Omron Sysmac Studio project 2.0_integration_1 (Sysmac Studio 1.54.0.64019, StandardProject)

# Controller new_Controller_0: NJ301-1100 version 1.14
Units and slaves: Node1 : NX-ECC201 (E001); Unit 1 : NX-PC0020 (N1); Unit 2 : NX-ID5442 (N2); Unit 3 : NX-PC0010 (N3); Unit 4 : NX-PC0020 (N4); Unit 5 : NX-OD5121 (N5); Unit 6 : NX-PC0010 (N6); Power Supply : NJ-Px3001; CPU : NJ301-1100; 0 [Unit 0] : CJ1W-AD041-V1 (J01); 1 [Unit 1] : CJ1W-DA041 (J02); 2 : CJ1W-ID211 (J03); 3 : CJ1W-OC211 (J04)
Task PrimaryTask (priority 4, period or condition 1000): Program0

VAR_GLOBAL
    Station_1B2 : BOOL;  (* Lifting Cylinder Down; at IOBus://rack#0/slot#2/Ch1_In/Ch1_In05; published *)
    Station_1B1 : BOOL;  (* Lifting Cylinder Up; at IOBus://rack#0/slot#2/Ch1_In/Ch1_In04; published *)
    Station_B5 : BOOL;  (* Workpiece Height Correct; at IOBus://rack#0/slot#2/Ch1_In/Ch1_In03; published *)
    Station_3S1 : BOOL;  (* arm_in_magazine; published *)
    Station_3S2 : BOOL;  (* arm_in_downstream; published *)
    Station_2B1 : BOOL;  (* Ejecting Cylinder Retracted; at IOBus://rack#0/slot#2/Ch1_In/Ch1_In06; published *)
    Panel_S1 : BOOL;  (* start_button; at IOBus://rack#0/slot#2/Ch1_In/Ch1_In08; published *)
    Panel_S2 : BOOL;  (* stop_button; at IOBus://rack#0/slot#2/Ch1_In/Ch1_In09; published *)
    Panel_S4 : BOOL;  (* reset_button; at IOBus://rack#0/slot#2/Ch1_In/Ch1_In11; published *)
    Station_1Y1 : BOOL;  (* Lift Down; at IOBus://rack#0/slot#3/Ch1_Out/Ch1_Out00; published *)
    Station_1Y2 : BOOL;  (* Lift Up; at IOBus://rack#0/slot#3/Ch1_Out/Ch1_Out01; published *)
    Station_2Y1 : BOOL;  (* Advance Ejecting Cylinder; at IOBus://rack#0/slot#3/Ch1_Out/Ch1_Out02; published *)
    Station_3Y1 : BOOL;  (* Air Cushion On; at IOBus://rack#0/slot#3/Ch1_Out/Ch1_Out03; published *)
    Station_3Y2 : BOOL;  (* arm_2_downstream; published *)
    Station_H1 : BOOL;  (* start light; at IOBus://rack#0/slot#3/Ch1_Out/Ch1_Out08; published *)
    Station_H2 : BOOL;  (* reset light; at IOBus://rack#0/slot#3/Ch1_Out/Ch1_Out09; published *)
    Panel_H3 : BOOL;  (* Q1 light; at IOBus://rack#0/slot#3/Ch1_Out/Ch1_Out10; published *)
    Panel_H4 : BOOL;  (* Q2 light; at IOBus://rack#0/slot#3/Ch1_Out/Ch1_Out11; published *)
    Station_1B1_in : BOOL;
    IP_FI : BOOL;  (* Succeeding Station Free; at IOBus://rack#0/slot#2/Ch1_In/Ch1_In07 *)
    Part_AV : BOOL;  (* Workpiece Available; at IOBus://rack#0/slot#2/Ch1_In/Ch1_In00 *)
    Station_B2 : BOOL;  (* Workpiece not black; at IOBus://rack#0/slot#2/Ch1_In/Ch1_In01 *)
    Station_B4 : BOOL;  (* Safety Through Beam; at IOBus://rack#0/slot#2/Ch1_In/Ch1_In02 *)
    IP_N_FO : BOOL;  (* Station Occupied; at IOBus://rack#0/slot#3/Ch1_Out/Ch1_Out07 *)
END_VAR

PROGRAM Program0
VAR
    FB_Panel_1 : FB_Panel;
    run_mode : BOOL;
    stop_mode : BOOL;
    reset_mode : BOOL;
    FB_Actuator_T1_1 : FB_Actuator_T1;
    timer_t1 : TON;
    error_mode : BOOL;
    FB_Actuator_T2_1 : FB_Actuator_T2;
    Piston : RS;
    error_ejec : BOOL;
    extend_piston : BOOL;
    workpiece_ready_set : BOOL;
    flip_flop_1 : RS;
    workpiece_ready : BOOL;
    workpiece_picked_up : BOOL;
    wait_for_piston : TON;
    Workpiece_Checker_1 : Workpiece_Checker;
    error_state : BOOL;
    error_suction : BOOL;
    error_t1 : BOOL;
    error_t2 : BOOL;
    rs1 : RS;
    rs2 : RS;
    rs3 : RS;
    e1 : BOOL;
    e2 : BOOL;
    e3 : BOOL;
    error_lift : BOOL;
    Control_T1_1 : Control_T1;
    error_q2_out : BOOL;
    Station_h3 : BOOL;
    Station_h4 : BOOL;
    FB_Receiver_1 : FB_Receiver;
    start_reciever : BOOL;
    stop_reciever : BOOL;
    reset_reciever : BOOL;
    next_ready : BOOL;
    start_button : BOOL;
    stop_button : BOOL;
    reset_button : BOOL;
    FB_Sender_1 : FB_Sender;
    need_piece : BOOL;
END_VAR
VAR_EXTERNAL
    Station_3S1 : BOOL;
    Panel_S2 : BOOL;
    Station_3Y2 : BOOL;
    Station_3S2 : BOOL;
    Panel_S1 : BOOL;
    Station_3Y1 : BOOL;
    Panel_S4 : BOOL;
    Station_H1 : BOOL;
    Station_H2 : BOOL;
    Panel_H4 : BOOL;
    Panel_H3 : BOOL;
    Station_1B2 : BOOL;
    Station_1B1 : BOOL;
    Station_1Y1 : BOOL;
    Station_2Y1 : BOOL;
    Station_2B1 : BOOL;
    Station_B4 : BOOL;
    Station_1Y2 : BOOL;
    Station_B2 : BOOL;
    Part_AV : BOOL;
    Station_B5 : BOOL;
    IP_FI : BOOL;
    IP_N_FO : BOOL;
END_VAR

(* Section Section0: ladder, written here as Structured Text *)

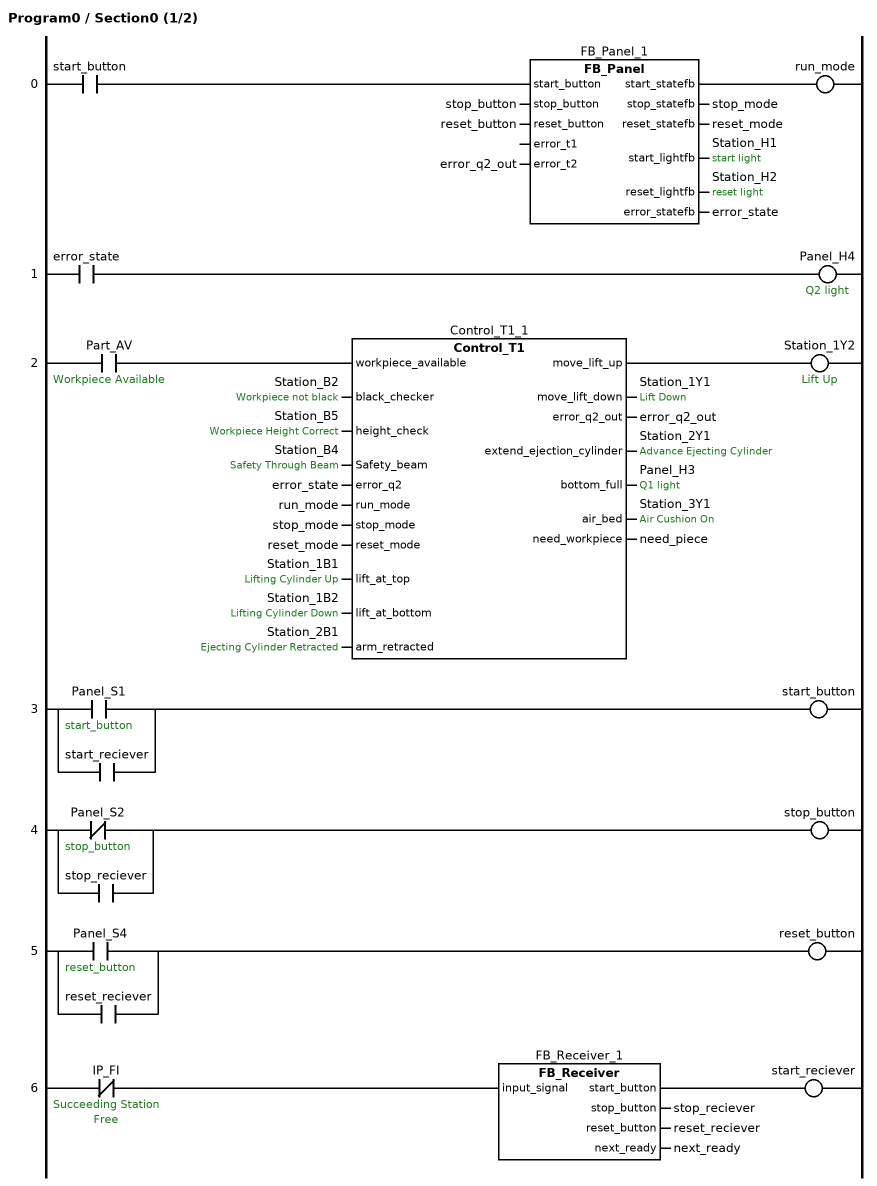
(* Rung 0 *)
FB_Panel_1(start_button := start_button, stop_button := stop_button, reset_button := reset_button, error_t2 := error_q2_out, stop_statefb => stop_mode, reset_statefb => reset_mode, start_lightfb => Station_H1, reset_lightfb => Station_H2, error_statefb => error_state);
run_mode := FB_Panel_1.start_statefb;
(* Rung 1 *)
Panel_H4 := error_state;
(* Rung 2 *)
Control_T1_1(workpiece_available := Part_AV, black_checker := Station_B2, height_check := Station_B5, Safety_beam := Station_B4, error_q2 := error_state, run_mode := run_mode, stop_mode := stop_mode, reset_mode := reset_mode, lift_at_top := Station_1B1, lift_at_bottom := Station_1B2, arm_retracted := Station_2B1, move_lift_down => Station_1Y1, error_q2_out => error_q2_out, extend_ejection_cylinder => Station_2Y1, bottom_full => Panel_H3, air_bed => Station_3Y1, need_workpiece => need_piece);
Station_1Y2 := Control_T1_1.move_lift_up;
(* Rung 3 *)
start_button := Panel_S1 OR start_reciever;
(* Rung 4 *)
stop_button := NOT Panel_S2 OR stop_reciever;
(* Rung 5 *)
reset_button := Panel_S4 OR reset_reciever;
(* Rung 6 *)
FB_Receiver_1(input_signal := NOT IP_FI, stop_button => stop_reciever, reset_button => reset_reciever, next_ready => next_ready);
start_reciever := FB_Receiver_1.start_button;

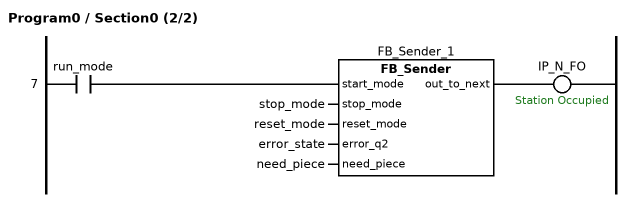
(* Rung 7 *)
FB_Sender_1(start_mode := run_mode, stop_mode := stop_mode, reset_mode := reset_mode, error_q2 := error_state, need_piece := need_piece);
IP_N_FO := FB_Sender_1.out_to_next;
END_PROGRAM

FUNCTION_BLOCK FB_Panel
VAR
    flip_flop : RS;
    flip_flop2 : RS;
    flip_flop_3 : RS;
    flip_flop3 : RS;
    stop_or_error : BOOL;
    error_q2 : BOOL;
    flip_flop4 : RS;
END_VAR
VAR_OUTPUT
    start_statefb : BOOL;
    stop_statefb : BOOL;
    reset_statefb : BOOL;
END_VAR
VAR_INPUT
    start_button : BOOL := False;
    stop_button : BOOL := False;
    reset_button : BOOL := False;
END_VAR
VAR_OUTPUT
    start_lightfb : BOOL;
    reset_lightfb : BOOL;
    error_statefb : BOOL;
END_VAR
VAR_INPUT
    error_t1 : BOOL;
    error_t2 : BOOL;
END_VAR
VAR_EXTERNAL
    Panel_H4 : BOOL;
END_VAR
(* ladder, written here as Structured Text *)

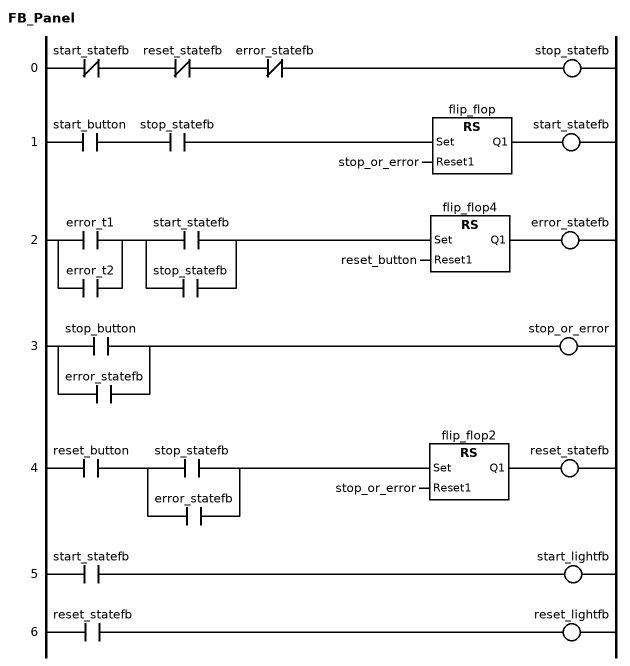
(* Rung 0 *)
stop_statefb := NOT start_statefb AND NOT reset_statefb AND NOT error_statefb;
(* Rung 1 *)
flip_flop(Set := start_button AND stop_statefb, Reset1 := stop_or_error);
start_statefb := flip_flop.Q1;
(* Rung 2 *)
flip_flop4(Set := (error_t1 OR error_t2) AND (start_statefb OR stop_statefb), Reset1 := reset_button);
error_statefb := flip_flop4.Q1;
(* Rung 3 *)
stop_or_error := stop_button OR error_statefb;
(* Rung 4 *)
flip_flop2(Set := reset_button AND (stop_statefb OR error_statefb), Reset1 := stop_or_error);
reset_statefb := flip_flop2.Q1;
(* Rung 5 *)
start_lightfb := start_statefb;
(* Rung 6 *)
reset_lightfb := reset_statefb;
END_FUNCTION_BLOCK

FUNCTION_BLOCK FB_Actuator_T2
VAR
    reset_to_home : BOOL;
    retract_ff : RS;
    extend_ff : RS;
    extend_t : TON;
    retract_t : TON;
    retract_err : BOOL;
    extend_err : BOOL;
    workpiece_lifted : BOOL;
    Workpiece_ejection : RS;
END_VAR
VAR_INPUT
    run_mode : BOOL;
    reset_mode : BOOL;
    stop_mode : BOOL;
    error_mode : BOOL;
END_VAR
VAR_OUTPUT
    retract_piston : BOOL;
    extend_piston : BOOL;
END_VAR
VAR_INPUT
    piston_retracted : BOOL;
    piston_extended : BOOL;
END_VAR
VAR_OUTPUT
    error_eject : BOOL;
END_VAR
VAR_INPUT
    Workpiece_ready : BOOL;
END_VAR
VAR_OUTPUT
    Mag_Empty_out : BOOL;
END_VAR
VAR_INPUT
    Mag_state : BOOL;
END_VAR
VAR_EXTERNAL
    Station_B4 : BOOL;
    Station_1B1 : BOOL;
    Station_1B2 : BOOL;
    Station_2Y1 : BOOL;
END_VAR
(* ladder, written here as Structured Text *)

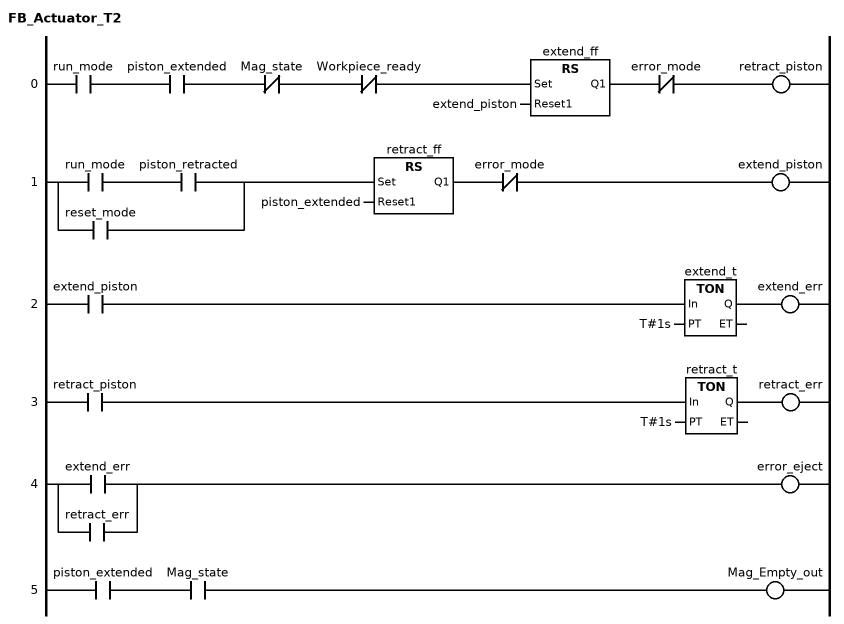
(* Rung 0 *)
extend_ff(Set := run_mode AND piston_extended AND NOT Mag_state AND NOT Workpiece_ready, Reset1 := extend_piston);
retract_piston := extend_ff.Q1 AND NOT error_mode;
(* Rung 1 *)
retract_ff(Set := (run_mode AND piston_retracted) OR reset_mode, Reset1 := piston_extended);
extend_piston := retract_ff.Q1 AND NOT error_mode;
(* Rung 2 *)
extend_t(In := extend_piston, PT := T#1s);
extend_err := extend_t.Q;
(* Rung 3 *)
retract_t(In := retract_piston, PT := T#1s);
retract_err := retract_t.Q;
(* Rung 4 *)
error_eject := extend_err OR retract_err;
(* Rung 5 *)
Mag_Empty_out := piston_extended AND Mag_state;
END_FUNCTION_BLOCK

FUNCTION_BLOCK Workpiece_Checker
VAR
    wait_for_piston : TON;
    flip_flop_1 : RS;
    workpiece_not_ready : BOOL;
END_VAR
VAR_INPUT
    reset_state : BOOL;
    workpiece_ready_set : BOOL;
    workpiece_picked_up : BOOL (* edge DownDirection *);
END_VAR
VAR_OUTPUT
    workpiece_ready : BOOL;
END_VAR
(* ladder, written here as Structured Text *)

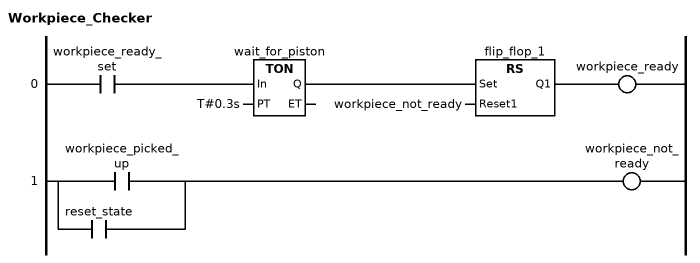
(* Rung 0 *)
wait_for_piston(In := workpiece_ready_set, PT := T#0.3s);
flip_flop_1(Set := wait_for_piston.Q, Reset1 := workpiece_not_ready);
workpiece_ready := flip_flop_1.Q1;
(* Rung 1 *)
workpiece_not_ready := workpiece_picked_up OR reset_state;
END_FUNCTION_BLOCK

FUNCTION_BLOCK FB_Actuator_T1
VAR
    flip_flop_1 : RS;
    flip_flop_2 : RS;
    reset_to_home : BOOL;
    timer_t1 : TON;
    flip_flop_3 : RS;
    timer_t2 : TON;
    flip_flop_4 : RS;
    error_toSub : BOOL;
    error_toHome : BOOL;
    middle_timer : AccumulationTimer;
    flip_flop_5 : RS;
    reset_middle : BOOL;
    flip_flop6 : RS;
    move_to_middle_from_home : BOOL;
    move_to_home : BOOL;
    move_to_middle_from_sub : BOOL;
    unknown_pos : BOOL;
    reset_vac_arm_to_sub : BOOL;
    timer_t3 : TON;
    t : TIME;
    unknown_pos_timer : TON;
    TOF_1 : TOF;
    move_to_sub : BOOL;
END_VAR
VAR_INPUT
    Arm_In_Mag_Pos : BOOL;
    Arm_In_Sub_Pos : BOOL;
    stop_mode : BOOL;
END_VAR
VAR_OUTPUT
    error_arm : BOOL;
    arm_to_sub : BOOL;
    arm_to_home : BOOL;
END_VAR
VAR_INPUT
    error_q2 : BOOL;
    set_move_to_sub : BOOL;
    set_move_to_home : BOOL;
    set_move_to_middle_from_home : BOOL;
    set_move_to_middle_from_sub : BOOL;
END_VAR
VAR_OUTPUT
    middle_pos : BOOL;
END_VAR
VAR_INPUT
    reset_mode : BOOL;
END_VAR
VAR_EXTERNAL
    Station_1B1 : BOOL;
END_VAR
(* ladder, written here as Structured Text *)

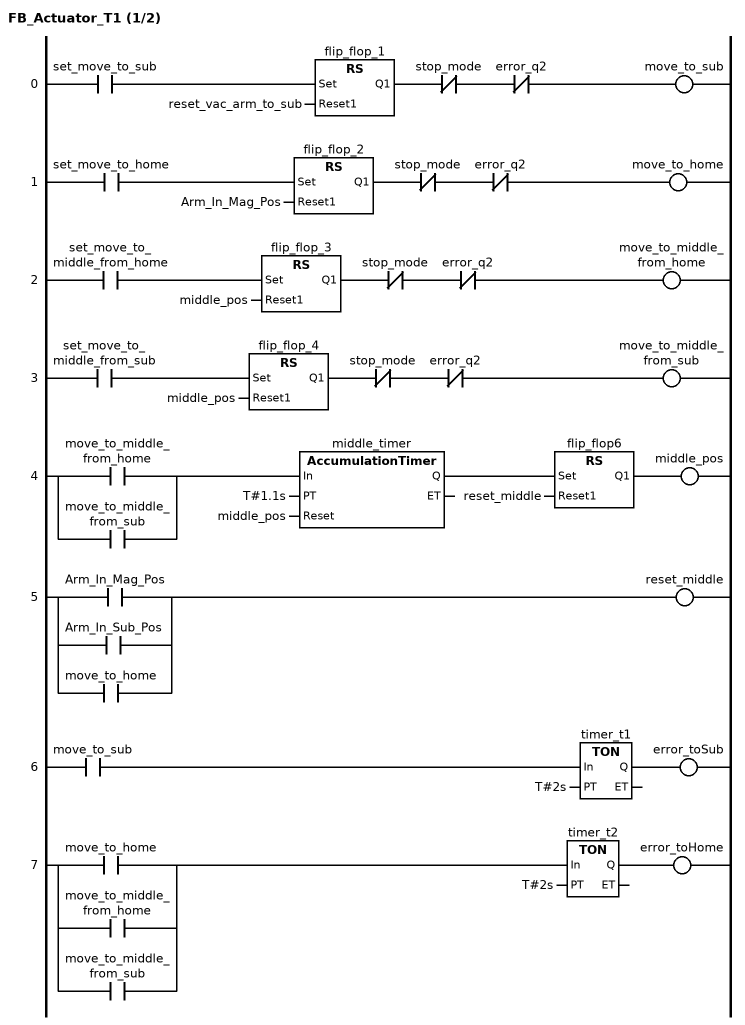
(* Rung 0 *)
flip_flop_1(Set := set_move_to_sub, Reset1 := reset_vac_arm_to_sub);
move_to_sub := flip_flop_1.Q1 AND NOT stop_mode AND NOT error_q2;
(* Rung 1 *)
flip_flop_2(Set := set_move_to_home, Reset1 := Arm_In_Mag_Pos);
move_to_home := flip_flop_2.Q1 AND NOT stop_mode AND NOT error_q2;
(* Rung 2 *)
flip_flop_3(Set := set_move_to_middle_from_home, Reset1 := middle_pos);
move_to_middle_from_home := flip_flop_3.Q1 AND NOT stop_mode AND NOT error_q2;
(* Rung 3 *)
flip_flop_4(Set := set_move_to_middle_from_sub, Reset1 := middle_pos);
move_to_middle_from_sub := flip_flop_4.Q1 AND NOT stop_mode AND NOT error_q2;
(* Rung 4 *)
middle_timer(In := move_to_middle_from_home OR move_to_middle_from_sub, PT := T#1.1s, Reset := middle_pos);
flip_flop6(Set := middle_timer.Q, Reset1 := reset_middle);
middle_pos := flip_flop6.Q1;
(* Rung 5 *)
reset_middle := Arm_In_Mag_Pos OR Arm_In_Sub_Pos OR move_to_home;
(* Rung 6 *)
timer_t1(In := move_to_sub, PT := T#2s);
error_toSub := timer_t1.Q;
(* Rung 7 *)
timer_t2(In := move_to_home OR move_to_middle_from_home OR move_to_middle_from_sub, PT := T#2s);
error_toHome := timer_t2.Q;

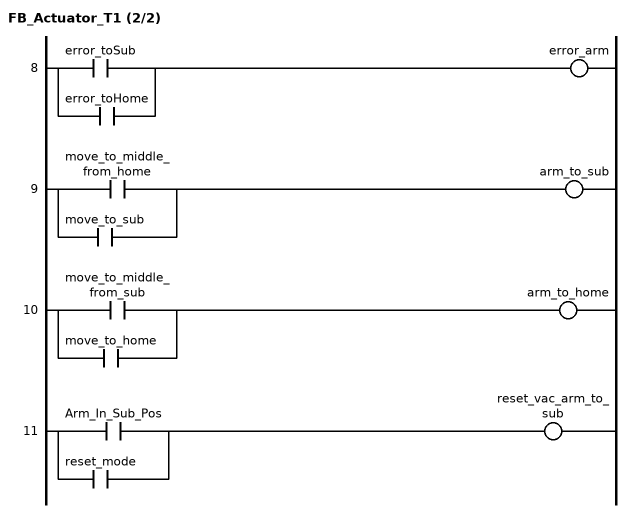
(* Rung 8 *)
error_arm := error_toSub OR error_toHome;
(* Rung 9 *)
arm_to_sub := move_to_middle_from_home OR move_to_sub;
(* Rung 10 *)
arm_to_home := move_to_middle_from_sub OR move_to_home;
(* Rung 11 *)
reset_vac_arm_to_sub := Arm_In_Sub_Pos OR reset_mode;
END_FUNCTION_BLOCK

FUNCTION_BLOCK Control_T1
VAR
    FB_Actuator_T1_1 : FB_Actuator_T1;
    set_move_lift_down : BOOL;
    set_move_lift_up : BOOL;
    lift_moved : BOOL;
    lift_move_rs : RS;
    wait_lift : BOOL;
    wait_t3_up : TON;
    wait_t3_down : TON;
    error_t3 : BOOL;
    error_lift : BOOL;
    reset_safety_beam : BOOL;
    Safety_beam_error_1 : BOOL;
    safety_timer : TON;
    Safety_beam_error_2 : BOOL;
    safet_beam_counter : CTU;
    safety_beam_error : BOOL;
    cnt : INT;
    TOF_safety_beam : TOF;
    safetybeam_TON : TON;
    t3_finished : BOOL;
    rs_output_top : RS;
    rs_output_bottom : RS;
    bottom_eject_counter : CTU;
    eject_top : BOOL;
    eject_bot : BOOL;
    reset_t3_ejector : BOOL;
    eject_bot_timer : TON;
    cnt2 : INT;
    actuator_T3 : BOOL;
    workpiece_carried_rs : RS;
    workpiece_carried : BOOL;
    cycle_complete : BOOL;
    reset_workpiece_carried : BOOL;
    r_trig_t3_cycle : R_TRIG;
    wait_lift_down : TON;
    eject_top_timer : TON;
    error_no_room_bottom : BOOL;
    rs_white_piece : RS;
    white_eject_bottom : BOOL;
    wait_lift_up : TON;
    rs_test_whiteandfull : RS;
    q2_full_bottom : BOOL;
    pulse_time_air_bed : TP;
    Control_T3_1 : control_T3;
    rs_error_t3 : RS;
    rs_error_safety_beam : RS;
    rs_error_lift : RS;
    test_error_t3 : BOOL;
    test_error_beam : BOOL;
    test_error_lift : BOOL;
    rs_bottom_full_error : RS;
    test_error_bottom : BOOL;
    TON_error_no_room_bottom : TON;
    delay_white_top : TON;
    reset_workpiece_carried_TP : TP;
    wait_T3 : CTU;
    cnt_actuator : INT;
    wait_workpiece_carried_TON : TON;
    request_workpiece_TON : TON;
END_VAR
VAR_INPUT
    workpiece_available : BOOL;
    black_checker : BOOL;
    height_check : BOOL;
    Safety_beam : BOOL;
    error_q2 : BOOL;
    run_mode : BOOL;
    stop_mode : BOOL;
    reset_mode : BOOL;
    lift_at_top : BOOL;
    lift_at_bottom : BOOL;
END_VAR
VAR_OUTPUT
    move_lift_up : BOOL;
    move_lift_down : BOOL;
    error_q2_out : BOOL;
    extend_ejection_cylinder : BOOL;
END_VAR
VAR_INPUT
    arm_retracted : BOOL;
END_VAR
VAR_OUTPUT
    bottom_full : BOOL;
    air_bed : BOOL;
    need_workpiece : BOOL;
END_VAR
VAR_EXTERNAL
    Station_1B1 : BOOL;
    Station_1B1_in : BOOL;
    Station_1B2 : BOOL;
    Station_B2 : BOOL;
END_VAR
VAR
    _e1 : R_TRIG;
    _e2 : R_TRIG;
END_VAR
(* ladder, written here as Structured Text *)

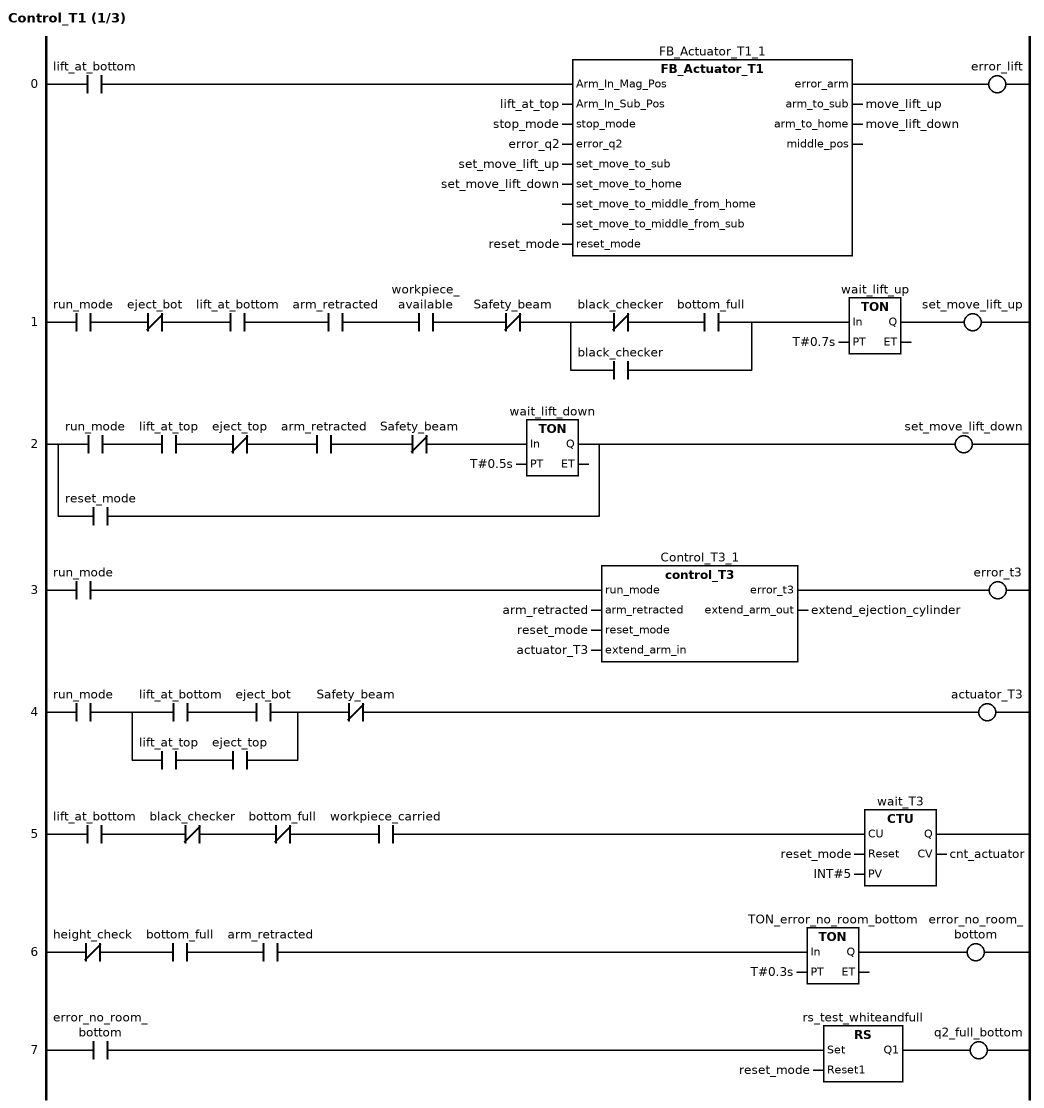
(* Rung 0 *)
FB_Actuator_T1_1(Arm_In_Mag_Pos := lift_at_bottom, Arm_In_Sub_Pos := lift_at_top, stop_mode := stop_mode, error_q2 := error_q2, set_move_to_sub := set_move_lift_up, set_move_to_home := set_move_lift_down, reset_mode := reset_mode, arm_to_sub => move_lift_up, arm_to_home => move_lift_down);
error_lift := FB_Actuator_T1_1.error_arm;
(* Rung 1 *)
wait_lift_up(In := run_mode AND NOT eject_bot AND lift_at_bottom AND arm_retracted AND workpiece_available AND NOT Safety_beam AND ((NOT black_checker AND bottom_full) OR black_checker), PT := T#0.7s);
set_move_lift_up := wait_lift_up.Q;
(* Rung 2 *)
wait_lift_down(In := run_mode AND lift_at_top AND NOT eject_top AND arm_retracted AND NOT Safety_beam, PT := T#0.5s);
set_move_lift_down := wait_lift_down.Q OR reset_mode;
(* Rung 3 *)
Control_T3_1(run_mode := run_mode, arm_retracted := arm_retracted, reset_mode := reset_mode, extend_arm_in := actuator_T3, extend_arm_out => extend_ejection_cylinder);
error_t3 := Control_T3_1.error_t3;
(* Rung 4 *)
actuator_T3 := run_mode AND ((lift_at_bottom AND eject_bot) OR (lift_at_top AND eject_top)) AND NOT Safety_beam;
(* Rung 5 *)
_e1(CLK := lift_at_bottom AND NOT black_checker AND NOT bottom_full AND workpiece_carried);
wait_T3(CU := _e1.Q, Reset := reset_mode, PV := INT#5, CV => cnt_actuator);
(* Rung 6 *)
TON_error_no_room_bottom(In := NOT height_check AND bottom_full AND arm_retracted, PT := T#0.3s);
error_no_room_bottom := TON_error_no_room_bottom.Q;
(* Rung 7 *)
rs_test_whiteandfull(Set := error_no_room_bottom, Reset1 := reset_mode);
q2_full_bottom := rs_test_whiteandfull.Q1;

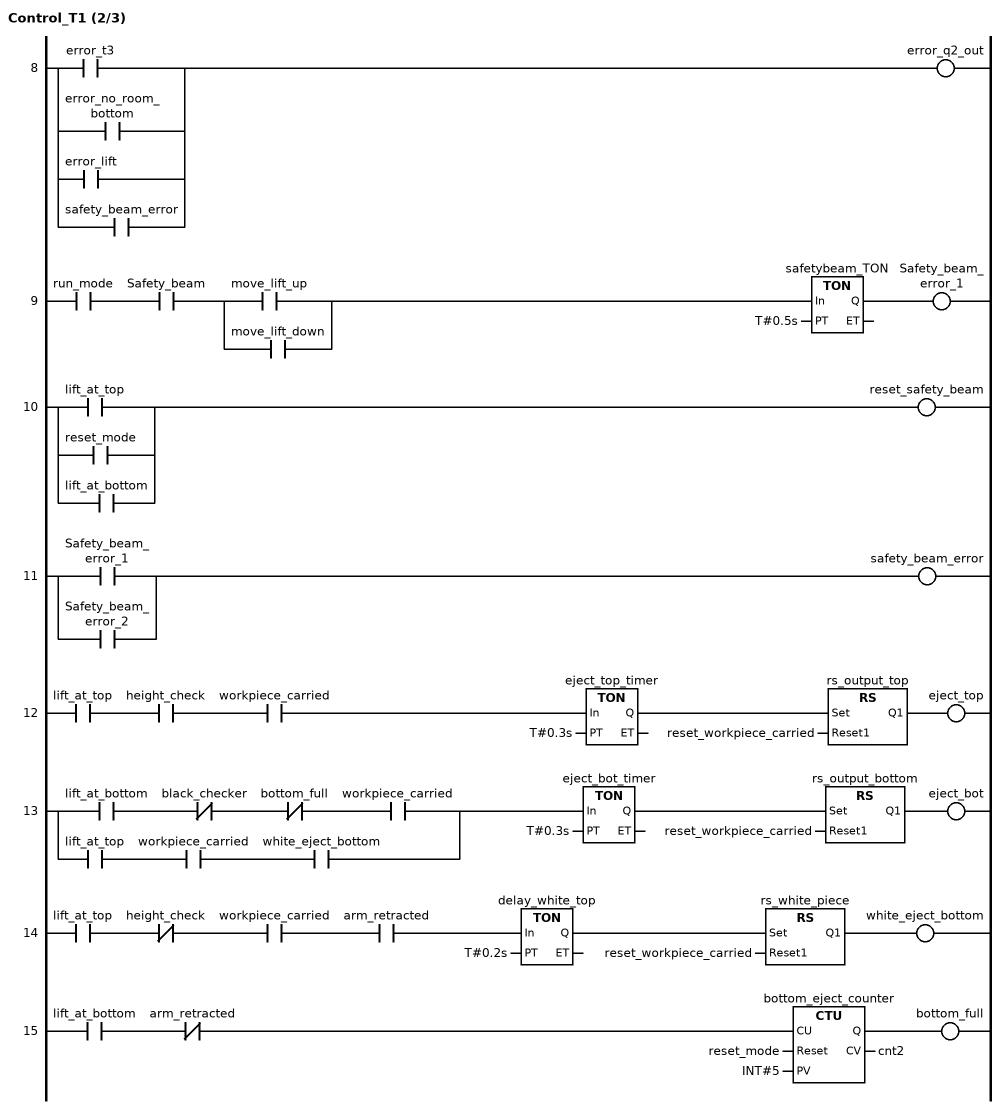
(* Rung 8 *)
error_q2_out := error_t3 OR error_no_room_bottom OR error_lift OR safety_beam_error;
(* Rung 9 *)
safetybeam_TON(In := run_mode AND Safety_beam AND (move_lift_up OR move_lift_down), PT := T#0.5s);
Safety_beam_error_1 := safetybeam_TON.Q;
(* Rung 10 *)
reset_safety_beam := lift_at_top OR reset_mode OR lift_at_bottom;
(* Rung 11 *)
safety_beam_error := Safety_beam_error_1 OR Safety_beam_error_2;
(* Rung 12 *)
eject_top_timer(In := lift_at_top AND height_check AND workpiece_carried, PT := T#0.3s);
rs_output_top(Set := eject_top_timer.Q, Reset1 := reset_workpiece_carried);
eject_top := rs_output_top.Q1;
(* Rung 13 *)
eject_bot_timer(In := (lift_at_bottom AND NOT black_checker AND NOT bottom_full AND workpiece_carried) OR (lift_at_top AND workpiece_carried AND white_eject_bottom), PT := T#0.3s);
rs_output_bottom(Set := eject_bot_timer.Q, Reset1 := reset_workpiece_carried);
eject_bot := rs_output_bottom.Q1;
(* Rung 14 *)
delay_white_top(In := lift_at_top AND NOT height_check AND workpiece_carried AND arm_retracted, PT := T#0.2s);
rs_white_piece(Set := delay_white_top.Q, Reset1 := reset_workpiece_carried);
white_eject_bottom := rs_white_piece.Q1;
(* Rung 15 *)
_e2(CLK := lift_at_bottom AND NOT arm_retracted);
bottom_eject_counter(CU := _e2.Q, Reset := reset_mode, PV := INT#5, CV => cnt2);
bottom_full := bottom_eject_counter.Q;

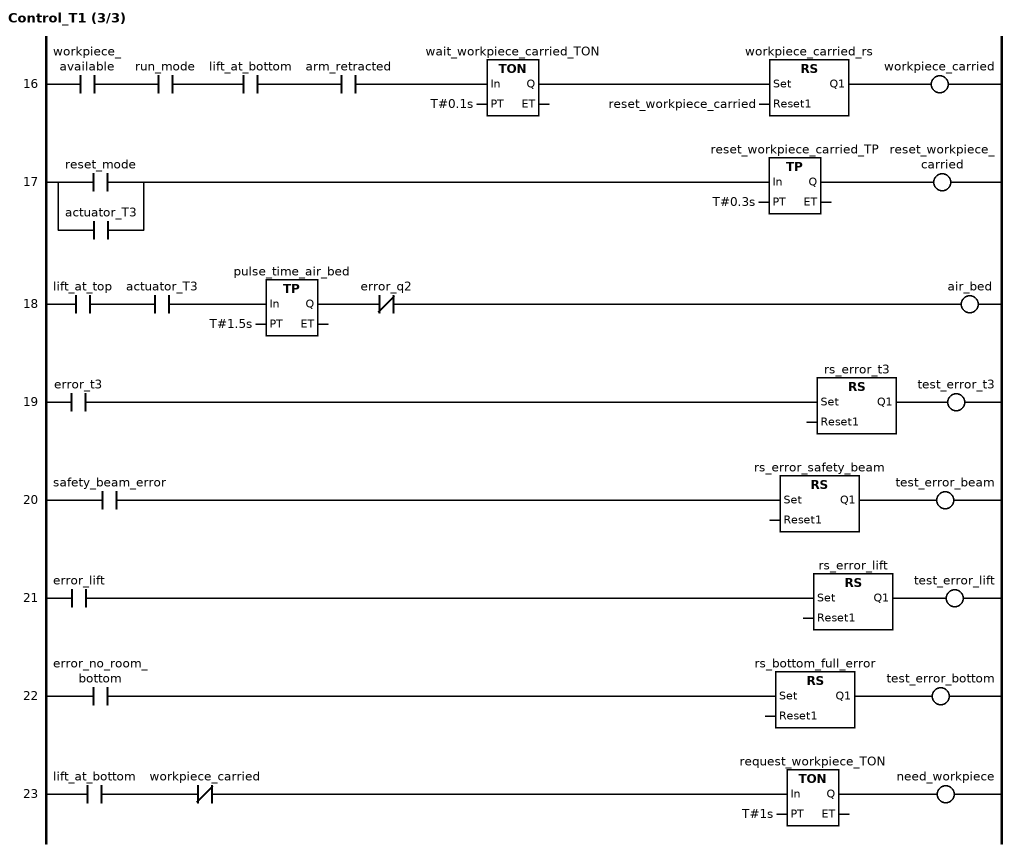
(* Rung 16 *)
wait_workpiece_carried_TON(In := workpiece_available AND run_mode AND lift_at_bottom AND arm_retracted, PT := T#0.1s);
workpiece_carried_rs(Set := wait_workpiece_carried_TON.Q, Reset1 := reset_workpiece_carried);
workpiece_carried := workpiece_carried_rs.Q1;
(* Rung 17 *)
reset_workpiece_carried_TP(In := reset_mode OR actuator_T3, PT := T#0.3s);
reset_workpiece_carried := reset_workpiece_carried_TP.Q;
(* Rung 18 *)
pulse_time_air_bed(In := lift_at_top AND actuator_T3, PT := T#1.5s);
air_bed := pulse_time_air_bed.Q AND NOT error_q2;
(* Rung 19 *)
rs_error_t3(Set := error_t3);
test_error_t3 := rs_error_t3.Q1;
(* Rung 20 *)
rs_error_safety_beam(Set := safety_beam_error);
test_error_beam := rs_error_safety_beam.Q1;
(* Rung 21 *)
rs_error_lift(Set := error_lift);
test_error_lift := rs_error_lift.Q1;
(* Rung 22 *)
rs_bottom_full_error(Set := error_no_room_bottom);
test_error_bottom := rs_bottom_full_error.Q1;
(* Rung 23 *)
request_workpiece_TON(In := lift_at_bottom AND NOT workpiece_carried, PT := T#1s);
need_workpiece := request_workpiece_TON.Q;
END_FUNCTION_BLOCK

FUNCTION_BLOCK FB_Actuator_T3
VAR
    TOF_1 : TOF;
    extend_arm_error_rs : RS;
    extend_arm_error_TON : TON;
    retract_arm : BOOL;
    Error_held_timer : AccumulationTimer;
    arm_extended_out : BOOL;
    reset_timer : BOOL;
    arm_out_timer : TON;
    arm_out_rs : RS;
    arm_extended_rs : RS;
    cycle_check_rs : RS;
    error_t3_1 : BOOL;
END_VAR
VAR_INPUT
    extend_arm_in : BOOL;
END_VAR
VAR_OUTPUT
    extend_arm_out : BOOL;
END_VAR
VAR_INPUT
    run_mode : BOOL;
    arm_retracted : BOOL;
END_VAR
VAR_OUTPUT
    error_t3 : BOOL;
END_VAR
VAR_INPUT
    reset_mode : BOOL;
    retract_arm_command : BOOL;
END_VAR
VAR_OUTPUT
    arm_extended : BOOL;
END_VAR
(* ladder, written here as Structured Text *)

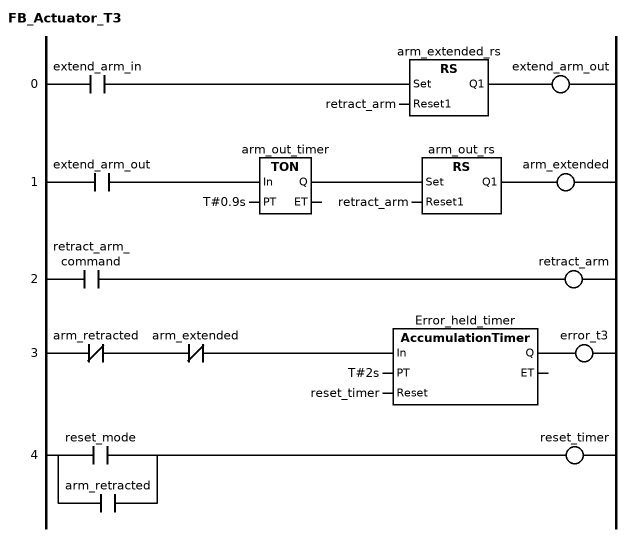
(* Rung 0 *)
arm_extended_rs(Set := extend_arm_in, Reset1 := retract_arm);
extend_arm_out := arm_extended_rs.Q1;
(* Rung 1 *)
arm_out_timer(In := extend_arm_out, PT := T#0.9s);
arm_out_rs(Set := arm_out_timer.Q, Reset1 := retract_arm);
arm_extended := arm_out_rs.Q1;
(* Rung 2 *)
retract_arm := retract_arm_command;
(* Rung 3 *)
Error_held_timer(In := NOT arm_retracted AND NOT arm_extended, PT := T#2s, Reset := reset_timer);
error_t3 := Error_held_timer.Q;
(* Rung 4 *)
reset_timer := reset_mode OR arm_retracted;
END_FUNCTION_BLOCK

FUNCTION_BLOCK control_T3
VAR
    FB_Actuator_T3_2 : FB_Actuator_T3;
    retract_arm : BOOL;
    arm_extended : BOOL;
    extend_arm_command : BOOL;
END_VAR
VAR_INPUT
    run_mode : BOOL;
    arm_retracted : BOOL;
    reset_mode : BOOL;
END_VAR
VAR_OUTPUT
    error_t3 : BOOL;
    extend_arm_out : BOOL;
END_VAR
VAR_INPUT
    extend_arm_in : BOOL;
END_VAR
(* ladder, written here as Structured Text *)

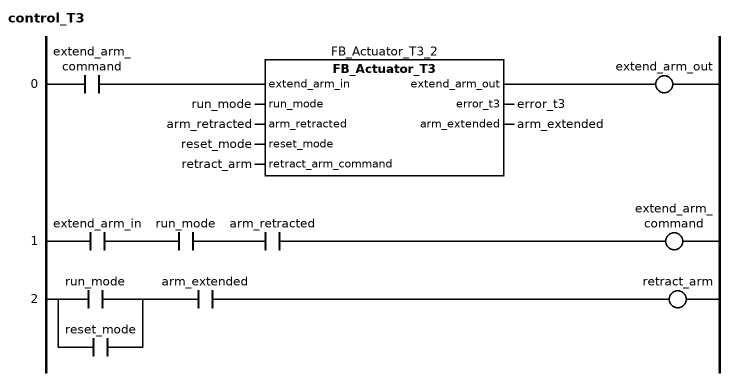
(* Rung 0 *)
FB_Actuator_T3_2(extend_arm_in := extend_arm_command, run_mode := run_mode, arm_retracted := arm_retracted, reset_mode := reset_mode, retract_arm_command := retract_arm, error_t3 => error_t3, arm_extended => arm_extended);
extend_arm_out := FB_Actuator_T3_2.extend_arm_out;
(* Rung 1 *)
extend_arm_command := extend_arm_in AND run_mode AND arm_retracted;
(* Rung 2 *)
retract_arm := (run_mode OR reset_mode) AND arm_extended;
END_FUNCTION_BLOCK

FUNCTION_BLOCK FB_Receiver
VAR
    pulse_length_timer : AccumulationTimer;
    reset_length : BOOL;
    pulse_length : TIME;
    timer_maxed : BOOL;
    wait_max_time : TON;
    max_time_signal : BOOL;
    start_counting_RS : RS;
    elapsed_time : TIME;
    pulse_length_comparison : FB_Reciever_Ladder_Logic;
    panel : BOOL;
END_VAR
VAR_OUTPUT
    start_button : BOOL;
    stop_button : BOOL;
    reset_button : BOOL;
    next_ready : BOOL;
END_VAR
VAR_INPUT
    input_signal : BOOL;
END_VAR
VAR_EXTERNAL
    Panel_H4 : BOOL;
    Panel_S2 : BOOL;
    Station_H2 : BOOL;
END_VAR
(* ladder, written here as Structured Text *)

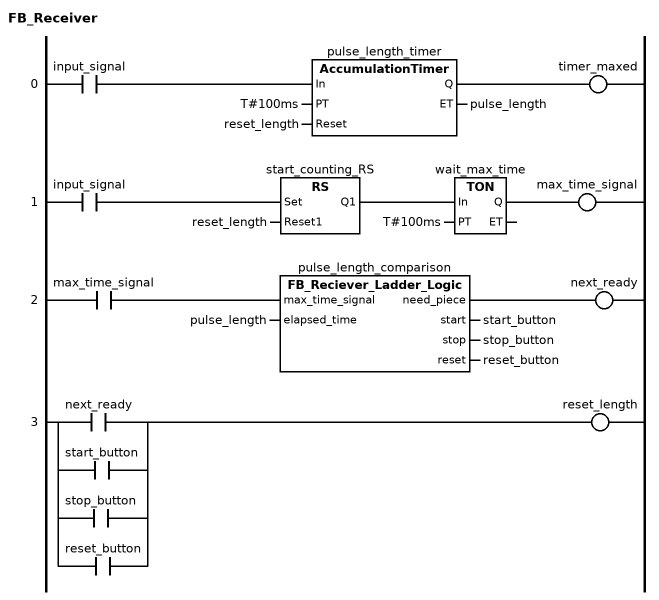
(* Rung 0 *)
pulse_length_timer(In := input_signal, PT := T#100ms, Reset := reset_length, ET => pulse_length);
timer_maxed := pulse_length_timer.Q;
(* Rung 1 *)
start_counting_RS(Set := input_signal, Reset1 := reset_length);
wait_max_time(In := start_counting_RS.Q1, PT := T#100ms);
max_time_signal := wait_max_time.Q;
(* Rung 2 *)
pulse_length_comparison(max_time_signal := max_time_signal, elapsed_time := pulse_length, start => start_button, stop => stop_button, reset => reset_button);
next_ready := pulse_length_comparison.need_piece;
(* Rung 3 *)
reset_length := next_ready OR start_button OR stop_button OR reset_button;
END_FUNCTION_BLOCK

FUNCTION_BLOCK FB_Reciever_Ladder_Logic
VAR_INPUT
    elapsed_time : TIME;
    max_time_signal : BOOL;
END_VAR
VAR_OUTPUT
    need_piece : BOOL;
    start : BOOL;
    stop : BOOL;
    reset : BOOL;
END_VAR
IF (max_time_signal) & (elapsed_time > T#70ms) THEN
	need_piece := TRUE;
	start := FALSE;
	stop := FALSE;
	reset := FALSE;
	
ELSIF (max_time_signal) & (elapsed_time > T#50ms)  THEN
	need_piece := FALSE;
	start := FALSE;
	stop := FALSE;
	reset := TRUE;

ELSIF (max_time_signal) & (elapsed_time > T#30ms)  THEN
	need_piece := FALSE;
	start := FALSE;
	stop := TRUE;
	reset := FALSE;
	
ELSIF (max_time_signal) & (elapsed_time >= T#0ms) THEN
	need_piece := FALSE;
	start := TRUE;
	stop := FALSE;
	reset := FALSE;
ELSE
	need_piece := FALSE;
	start := FALSE;
	stop := FALSE;
	reset := FALSE;

END_IF;
	
END_FUNCTION_BLOCK

FUNCTION_BLOCK FB_Sender
VAR
    start_mode_pulse : BOOL;
    stop_mode_pulse : BOOL;
    reset_mode_pulse : BOOL;
    start_pulse : TP;
    stop_pulse : TP;
    reset_pulse : TP;
    T : TIME;
    np_pulse_t : TP;
    np_pulse : BOOL;
    TON_need_piece : TON;
    et1 : TIME;
    et2 : TIME;
    et3 : TIME;
    et4 : TIME;
    test_stop_pulse : AccumulationTimer;
    et5 : TIME;
    stop_signal_wait : BOOL;
    start_signal_wait : BOOL;
    reset_signal_wait : BOOL;
    stop_signal_TP : TP;
    start_signal_TP : TP;
    reset_signal_TP : TP;
    wait_need_piece : TON;
END_VAR
VAR_INPUT
    start_mode : BOOL;
    stop_mode : BOOL;
    reset_mode : BOOL;
    error_q2 : BOOL;
    need_piece : BOOL;
END_VAR
VAR_OUTPUT
    out_to_next : BOOL;
END_VAR
(* ladder, written here as Structured Text *)

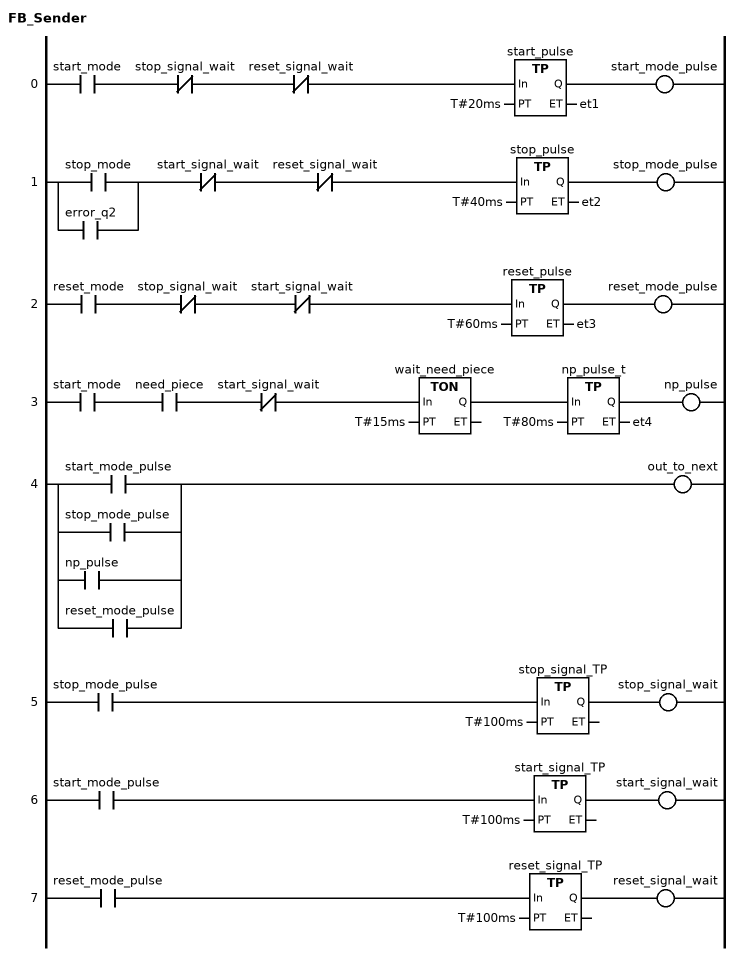
(* Rung 0 *)
start_pulse(In := start_mode AND NOT stop_signal_wait AND NOT reset_signal_wait, PT := T#20ms, ET => et1);
start_mode_pulse := start_pulse.Q;
(* Rung 1 *)
stop_pulse(In := (stop_mode OR error_q2) AND NOT start_signal_wait AND NOT reset_signal_wait, PT := T#40ms, ET => et2);
stop_mode_pulse := stop_pulse.Q;
(* Rung 2 *)
reset_pulse(In := reset_mode AND NOT stop_signal_wait AND NOT start_signal_wait, PT := T#60ms, ET => et3);
reset_mode_pulse := reset_pulse.Q;
(* Rung 3 *)
wait_need_piece(In := start_mode AND need_piece AND NOT start_signal_wait, PT := T#15ms);
np_pulse_t(In := wait_need_piece.Q, PT := T#80ms, ET => et4);
np_pulse := np_pulse_t.Q;
(* Rung 4 *)
out_to_next := start_mode_pulse OR stop_mode_pulse OR np_pulse OR reset_mode_pulse;
(* Rung 5 *)
stop_signal_TP(In := stop_mode_pulse, PT := T#100ms);
stop_signal_wait := stop_signal_TP.Q;
(* Rung 6 *)
start_signal_TP(In := start_mode_pulse, PT := T#100ms);
start_signal_wait := start_signal_TP.Q;
(* Rung 7 *)
reset_signal_TP(In := reset_mode_pulse, PT := T#100ms);
reset_signal_wait := reset_signal_TP.Q;
END_FUNCTION_BLOCK